{attribute 'GeneratedUsingTerminal: EK1122-0000-0018'}
{attribute addProperty BoxType "EK1122-0000-0018"}
{attribute addProperty Id "Beckhoff_ELM31xxsub_EK1100EK1100_1FC0878B2"}
{attribute addProperty CRC "3712570752"}
{attribute addProperty Size "2"}
TYPE Beckhoff_ELM31xxEK1122_DD495580 EXTENDS EK1122_1FC0878B :
STRUCT
	{attribute addProperty Name "Beckhoff ELM31xxsub EK1100"}
	{attribute addProperty PreviousPort "Beckhoff ELM31xxEK1122 : D"}
	Beckhoff_ELM31xxsub_EK1100 : EK1100_1FC0878B;
END_STRUCT
END_TYPE

(* stored: Version 1.2.0.0, ProductVersion 3.1.4024.9
   DUT Beckhoff_ELM31xxEK1122_DD495580: Id {aded55f7-ea4c-4cb3-96fc-e6a4a15719be} *)
